Staubli VAL3: onInsert.pgx

public program onInsert(string& x_sItem[])
  local string l_sEvent
  local num i
  local num l_nSize
  local string l_sMessage
  local num l_nKey
  local bool l_bFound
begin
  cls()
  call use:setView(false)
  call use:setSizeList(19,0,19,11)
  //
  // Prog
  //
  call use:listcreate("SUB")
  //
  call getSize(l_nSize)
  // refresh the list
  for i=0 to l_nSize-1
    call get(l_sEvent,i)
    if l_sEvent!=""
      // check it
        call use:listadd(l_sEvent)
    endIf
  endFor
  call use:listupdate(0)
  call language:message(l_sMessage,60)
  call use:typeLen(0,13,l_sMessage,40)
  do
    l_nKey=get()
    call use:listevent(l_nKey,i,x_sItem)
  until l_nKey==270 or l_nKey==255
  if l_nKey==255
    x_sItem=""
  endIf
end
